(* CODESYS project IoDrvSoundDemo.project

Project tree, tasks and I/O mapping:
  Device : CODESYS Control Win V3, 3S - Smart Software Solutions GmbH, order no. 305021, version 3.5.9.0
    application Application
      libraries: Standard, * (System); Analyzation, * (System); IecSfc, * (System)
      task Task (cyclic, interval t#20ms, priority 1) calls Main_PRG
      program Main_PRG [ST]
      visualisation MainVisu
      Function Blocks/
        function block JukeBox [ST]
      Enums/
        data type STATE
      GlobalVariables/
        global variables HAENSCHEN_KLEIN
        global variables FUER_ELISE
        global variables X_MAX
        global variables MUSICAL_SYMBOLS
      Structs/
        data type NOTE
      VisElements/
        visualisation Piano
        visualisation JukeBox
        image pool ImagePool
    SoundCard : SoundCard, Sound Company, version 3.3.0.0
        output ding : BOOL  // SoundOutput.Byte0.Bit0
        output cord : BOOL  // SoundOutput.Byte0.Bit1
        output chimes : BOOL  // SoundOutput.Byte0.Bit2
        output notify : BOOL  // SoundOutput.Byte0.Bit3
        output ringout : BOOL  // SoundOutput.Byte0.Bit4
        output tada : BOOL  // SoundOutput.Byte0.Bit5
        output _type : BOOL  // SoundOutput.Byte0.Bit6
        output newmail : BOOL  // SoundOutput.Byte0.Bit7
        output C : BOOL  // SoundOutput.Byte1.Bit0
        output Cis : BOOL  // SoundOutput.Byte1.Bit1
        output D : BOOL  // SoundOutput.Byte1.Bit2
        output Dis : BOOL  // SoundOutput.Byte1.Bit3
        output E : BOOL  // SoundOutput.Byte1.Bit4
        output F : BOOL  // SoundOutput.Byte1.Bit5
        output Fis : BOOL  // SoundOutput.Byte1.Bit6
        output G : BOOL  // SoundOutput.Byte1.Bit7
        output Gis : BOOL  // SoundOutput.Byte2.Bit0
        output A : BOOL  // SoundOutput.Byte2.Bit1
        output Ais : BOOL  // SoundOutput.Byte2.Bit2
        output H : BOOL  // SoundOutput.Byte2.Bit3
        output C_ : BOOL  // SoundOutput.Byte2.Bit4
        output Cis_ : BOOL  // SoundOutput.Byte2.Bit5
        output D_ : BOOL  // SoundOutput.Byte2.Bit6
        output Dis_ : BOOL  // SoundOutput.Byte2.Bit7
        output E_ : BOOL  // SoundOutput.Byte3.Bit0
        output F_ : BOOL  // SoundOutput.Byte3.Bit1
        output Fis_ : BOOL  // SoundOutput.Byte3.Bit2
        output G_ : BOOL  // SoundOutput.Byte3.Bit3
        output Gis_ : BOOL  // SoundOutput.Byte3.Bit4
        output A_ : BOOL  // SoundOutput.Byte3.Bit5
        output Ais_ : BOOL  // SoundOutput.Byte3.Bit6
        output H_ : BOOL  // SoundOutput.Byte3.Bit7
        unmapped channels: SoundOutput
  text list GlobalTextList
  5ce3da45-db07-42e7-a21c-a00fff4ed8f6|files\Jukebox\Fifties_jukebox.png
  5ce3da45-db07-42e7-a21c-a00fff4ed8f6|files\Jukebox\Fifties_jukebox9.png
  5ce3da45-db07-42e7-a21c-a00fff4ed8f6|files\Jukebox\Fifties_jukebox10.png
  5ce3da45-db07-42e7-a21c-a00fff4ed8f6|files\Jukebox\Fifties_jukebox11.png
  5ce3da45-db07-42e7-a21c-a00fff4ed8f6|files\Jukebox\Fifties_jukebox12.png
  5ce3da45-db07-42e7-a21c-a00fff4ed8f6|files\Jukebox\Fifties_jukebox13.png
  5ce3da45-db07-42e7-a21c-a00fff4ed8f6|files\Jukebox\Fifties_jukebox_1.png
  5ce3da45-db07-42e7-a21c-a00fff4ed8f6|files\Jukebox\Fifties_jukebox_2.png
  5ce3da45-db07-42e7-a21c-a00fff4ed8f6|files\Jukebox\Fifties_jukebox3.png
  5ce3da45-db07-42e7-a21c-a00fff4ed8f6|files\Jukebox\Fifties_jukebox4.png
  5ce3da45-db07-42e7-a21c-a00fff4ed8f6|files\Jukebox\Fifties_jukebox5.png
  5ce3da45-db07-42e7-a21c-a00fff4ed8f6|files\Jukebox\Fifties_jukebox6.png
  5ce3da45-db07-42e7-a21c-a00fff4ed8f6|files\Jukebox\Fifties_jukebox7.png
  5ce3da45-db07-42e7-a21c-a00fff4ed8f6|files\Jukebox\Fifties_jukebox8.png
*)

// Device/Application/Enums/STATE
// Each value represents a state which the program can have
{attribute 'qualified_only'}
TYPE STATE :
(
	PIANO := 0,			// change to Piano mode
	MUTE,				// No sound will be played 
	FUER_ELISE,			// play 'Für Elise' from Ludwig van Beethoven
	HAENSCHEN_KLEIN,	// play 'Hänschen klein' a German folk song from Franz Wiedemann 
	MERRY_XMAS,			// play 'We Wish You a Merry Christmas' 
	JUKE,				// change to Jukebox mode
	WAITING				// waiting for another command
);
END_TYPE

// Device/Application/Structs/NOTE
// This structure represents a note that can be played by the program
TYPE NOTE :
STRUCT
	tLength	: TIME;				// reflects duration of a note
	pNote	: POINTER TO BYTE;	// byte address of the output channel
	iBit	: INT;				// Offset from the output byte that addresses the sound
END_STRUCT
END_TYPE

// Device/Application/GlobalVariables/HAENSCHEN_KLEIN
// Hänschen klein - Franz Wiedemann
VAR_GLOBAL
	HAENSCHEN : ARRAY[0..31] OF NOTE := [
		(************ Takt01 ***************************)
		(	tLength:= 	T#500MS ,
			pNote :=	ADR(IoConfig_Globals_Mapping.G),
			iBit	:= 7
		),
		(	tLength:= 	T#450MS ,
			pNote :=	ADR(IoConfig_Globals_Mapping.E),
			iBit	:= 4
		),
		(	tLength:= 	T#50MS ,
			pNote :=	ADR(MUSICAL_SYMBOLS.xPause),
			iBit	:= 0
		),
		(	tLength:= 	T#1000MS ,
			pNote :=	ADR(IoConfig_Globals_Mapping.E),
			iBit	:= 4
		),
		(************ Takt02 ***************************)
		(	tLength:= 	T#500MS ,
			pNote :=	ADR(IoConfig_Globals_Mapping.F),
			iBit	:= 5
		),
		(	tLength:= 	T#450MS ,
			pNote :=	ADR(IoConfig_Globals_Mapping.D),
			iBit	:= 2
		),
		(	tLength:= 	T#50MS ,
			pNote :=	ADR(MUSICAL_SYMBOLS.xPause),
			iBit	:= 0
		),
		(	tLength:= 	T#1000MS ,
			pNote :=	ADR(IoConfig_Globals_Mapping.D),
			iBit	:= 2
		),
		(************ Takt03 ***************************)
		(	tLength:= 	T#500MS ,
			pNote :=	ADR(IoConfig_Globals_Mapping.C),
			iBit	:= 0
		),
		(	tLength:= 	T#500MS ,
			pNote :=	ADR(IoConfig_Globals_Mapping.D),
			iBit	:= 2
		),
		(	tLength:= 	T#500MS ,
			pNote :=	ADR(IoConfig_Globals_Mapping.E),
			iBit	:= 4
		),
		(	tLength:= 	T#500MS ,
			pNote :=	ADR(IoConfig_Globals_Mapping.F),
			iBit	:= 5
		),
		(************ Takt04 ***************************)
		(	tLength:= 	T#450MS ,
			pNote :=	ADR(IoConfig_Globals_Mapping.G),
			iBit	:= 7
		),
		(	tLength:= 	T#50MS ,
			pNote :=	ADR(MUSICAL_SYMBOLS.xPause),
			iBit	:= 0
		),
		(	tLength:= 	T#450MS ,
			pNote :=	ADR(IoConfig_Globals_Mapping.G),
			iBit	:= 7
		),
		(	tLength:= 	T#50MS ,
			pNote :=	ADR(MUSICAL_SYMBOLS.xPause),
			iBit	:= 0
		),
		(	tLength:= 	T#1000MS ,
			pNote :=	ADR(IoConfig_Globals_Mapping.G),
			iBit	:= 7
		),
		(************ Takt05 ***************************)
		(	tLength:= 	T#50MS ,
			pNote :=	ADR(MUSICAL_SYMBOLS.xPause),
			iBit	:= 0
		),
		(	tLength:= 	T#450MS ,
			pNote :=	ADR(IoConfig_Globals_Mapping.G),
			iBit	:= 7
		),
		(	tLength:= 	T#450MS ,
			pNote :=	ADR(IoConfig_Globals_Mapping.E),
			iBit	:= 4
		),
		(	tLength:= 	T#50MS ,
			pNote :=	ADR(MUSICAL_SYMBOLS.xPause),
			iBit	:= 0
		),
		(	tLength:= 	T#1000MS ,
			pNote :=	ADR(IoConfig_Globals_Mapping.E),
			iBit	:= 4
		),
		(************ Takt06 ***************************)
		(	tLength:= 	T#500MS ,
			pNote :=	ADR(IoConfig_Globals_Mapping.F),
			iBit	:= 5
		),
		(	tLength:= 	T#450MS ,
			pNote :=	ADR(IoConfig_Globals_Mapping.D),
			iBit	:= 2
		),
		(	tLength:= 	T#50MS ,
			pNote :=	ADR(MUSICAL_SYMBOLS.xPause),
			iBit	:= 0
		),
		(	tLength:= 	T#1000MS ,
			pNote :=	ADR(IoConfig_Globals_Mapping.D),
			iBit	:= 2
		),
		(************ Takt07 ***************************)
		(	tLength:= 	T#500MS ,
			pNote :=	ADR(IoConfig_Globals_Mapping.C),
			iBit	:= 0
		),
		(	tLength:= 	T#500MS ,
			pNote :=	ADR(IoConfig_Globals_Mapping.E),
			iBit	:= 4
		),
		(	tLength:= 	T#450MS ,
			pNote :=	ADR(IoConfig_Globals_Mapping.G),
			iBit	:= 7
		),
		(	tLength:= 	T#50MS ,
			pNote :=	ADR(MUSICAL_SYMBOLS.xPause),
			iBit	:= 0
		),
		(	tLength:= 	T#500MS ,
			pNote :=	ADR(IoConfig_Globals_Mapping.G),
			iBit	:= 7
		),
		(************ Takt08 ***************************)
		(	tLength:= 	T#4000MS ,
			pNote :=	ADR(IoConfig_Globals_Mapping.C),
			iBit	:= 0
		)
	];
		
END_VAR

// Device/Application/GlobalVariables/FUER_ELISE
// Für Elise - Ludwig van Beethoven

VAR_GLOBAL
	ELISE : ARRAY[0..149] OF NOTE := [
		(************ Auftakt ***************************)
		(	tLength:= 	T#250MS ,
			pNote :=	ADR(IoConfig_Globals_Mapping.E_),
			iBit	:= 0
		),
		(	tLength:= 	T#250MS ,
			pNote :=	ADR(IoConfig_Globals_Mapping.Dis_),
			iBit	:= 7
		),
		(************ Takt01 ***************************)
		(	tLength:= 	T#250MS ,
			pNote :=	ADR(IoConfig_Globals_Mapping.E_),
			iBit	:= 0
		),
		(	tLength:= 	T#250MS ,
			pNote :=	ADR(IoConfig_Globals_Mapping.Dis_),
			iBit	:= 7
		),
		(	tLength:= 	T#250MS ,
			pNote :=	ADR(IoConfig_Globals_Mapping.E_),
			iBit	:= 0
		),
		(	tLength:= 	T#250MS ,
			pNote :=	ADR(IoConfig_Globals_Mapping.H),
			iBit	:= 3
		),
		(	tLength:= 	T#250MS ,
			pNote :=	ADR(IoConfig_Globals_Mapping.D_),
			iBit	:= 6
		),
		(	tLength:= 	T#250MS ,
			pNote :=	ADR(IoConfig_Globals_Mapping.C_),
			iBit	:= 4
		),
		(************ Takt02 ***************************)
		(	tLength:= 	T#500MS ,
			pNote :=	ADR(IoConfig_Globals_Mapping.A),
			iBit	:= 1
		),
		(	tLength:= 	T#250MS ,
			pNote :=	ADR(MUSICAL_SYMBOLS.xPause),
			iBit	:= 0
		),
		(	tLength:= 	T#250MS ,
			pNote :=	ADR(IoConfig_Globals_Mapping.C),
			iBit	:= 0
		),
		(	tLength:= 	T#250MS ,
			pNote :=	ADR(IoConfig_Globals_Mapping.E),
			iBit	:= 4
		),
		(	tLength:= 	T#250MS ,
			pNote :=	ADR(IoConfig_Globals_Mapping.A),
			iBit	:= 1
		),
		(************ Takt03 ***************************)
		(	tLength:= 	T#500MS ,
			pNote :=	ADR(IoConfig_Globals_Mapping.H),
			iBit	:= 3
		),
		(	tLength:= 	T#250MS ,
			pNote :=	ADR(MUSICAL_SYMBOLS.xPause),
			iBit	:= 0
		),
		(	tLength:= 	T#250MS ,
			pNote :=	ADR(IoConfig_Globals_Mapping.E),
			iBit	:= 4
		),
		(	tLength:= 	T#250MS ,
			pNote :=	ADR(IoConfig_Globals_Mapping.Gis),
			iBit	:= 0
		),
		(	tLength:= 	T#250MS ,
			pNote :=	ADR(IoConfig_Globals_Mapping.H),
			iBit	:= 3
		),
		(************ Takt04  ***************************)
		(	tLength:= 	T#500MS ,
			pNote :=	ADR(IoConfig_Globals_Mapping.C_),
			iBit	:= 4
		), 
		(	tLength:= 	T#250MS ,
			pNote :=	ADR(MUSICAL_SYMBOLS.xPause),
			iBit	:= 0
		),
		(	tLength:= 	T#250MS ,
			pNote :=	ADR(IoConfig_Globals_Mapping.E),
			iBit	:= 4
		),
		(	tLength:= 	T#250MS ,
			pNote :=	ADR(IoConfig_Globals_Mapping.E_),
			iBit	:= 0
		),
		(	tLength:= 	T#250MS ,
			pNote :=	ADR(IoConfig_Globals_Mapping.Dis_),
			iBit	:= 7
		),
		(************ Takt05 ***************************)
		(	tLength:= 	T#250MS ,
			pNote :=	ADR(IoConfig_Globals_Mapping.E_),
			iBit	:= 0
		),
		(	tLength:= 	T#250MS ,
			pNote :=	ADR(IoConfig_Globals_Mapping.Dis_),
			iBit	:= 7
		),
		(	tLength:= 	T#250MS ,
			pNote :=	ADR(IoConfig_Globals_Mapping.E_),
			iBit	:= 0
		),
		(	tLength:= 	T#250MS ,
			pNote :=	ADR(IoConfig_Globals_Mapping.H),
			iBit	:= 3
		),
		(	tLength:= 	T#250MS ,
			pNote :=	ADR(IoConfig_Globals_Mapping.D_),
			iBit	:= 6
		),
		(	tLength:= 	T#250MS ,
			pNote :=	ADR(IoConfig_Globals_Mapping.C_),
			iBit	:= 4
		),
		(************ Takt06 ***************************)
		(	tLength:= 	T#500MS ,
			pNote :=	ADR(IoConfig_Globals_Mapping.A),
			iBit	:= 1
		),
		(	tLength:= 	T#250MS ,
			pNote :=	ADR(MUSICAL_SYMBOLS.xPause),
			iBit	:= 0
		),
		(	tLength:= 	T#250MS ,
			pNote :=	ADR(IoConfig_Globals_Mapping.C),
			iBit	:= 0
		),
		(	tLength:= 	T#250MS ,
			pNote :=	ADR(IoConfig_Globals_Mapping.E),
			iBit	:= 4
		),
		(	tLength:= 	T#250MS ,
			pNote :=	ADR(IoConfig_Globals_Mapping.A),
			iBit	:= 1
		),
		(************ Takt07 ***************************)
		(	tLength:= 	T#500MS ,
			pNote :=	ADR(IoConfig_Globals_Mapping.H),
			iBit	:= 3
		),
		(	tLength:= 	T#50MS ,
			pNote :=	ADR(MUSICAL_SYMBOLS.xPause),
			iBit	:= 0
		),
		(	tLength:= 	T#200MS ,
			pNote :=	ADR(IoConfig_Globals_Mapping.E),
			iBit	:= 4
		),
		(	tLength:= 	T#250MS ,
			pNote :=	ADR(IoConfig_Globals_Mapping.C_),
			iBit	:= 4
		),
		(	tLength:= 	T#250MS ,
			pNote :=	ADR(IoConfig_Globals_Mapping.H),
			iBit	:= 3
		),
		(************ Takt08 ****************************)
		(	tLength:= 	T#1000MS ,
			pNote :=	ADR(IoConfig_Globals_Mapping.A),
			iBit	:= 1
		),
		(	tLength:= 	T#250MS ,
			pNote :=	ADR(IoConfig_Globals_Mapping.E_),
			iBit	:= 0
		),
		(	tLength:= 	T#250MS ,
			pNote :=	ADR(IoConfig_Globals_Mapping.Dis_),
			iBit	:= 7
		),
		(************ Takt09 ***************************)
		(	tLength:= 	T#250MS ,
			pNote :=	ADR(IoConfig_Globals_Mapping.E_),
			iBit	:= 0
		),
		(	tLength:= 	T#250MS ,
			pNote :=	ADR(IoConfig_Globals_Mapping.Dis_),
			iBit	:= 7
		),
		(	tLength:= 	T#250MS ,
			pNote :=	ADR(IoConfig_Globals_Mapping.E_),
			iBit	:= 0
		),
		(	tLength:= 	T#250MS ,
			pNote :=	ADR(IoConfig_Globals_Mapping.H),
			iBit	:= 3
		),
		(	tLength:= 	T#250MS ,
			pNote :=	ADR(IoConfig_Globals_Mapping.D_),
			iBit	:= 6
		),
		(	tLength:= 	T#250MS ,
			pNote :=	ADR(IoConfig_Globals_Mapping.C_),
			iBit	:= 4
		),
		(************ Takt10 ***************************)
		(	tLength:= 	T#500MS ,
			pNote :=	ADR(IoConfig_Globals_Mapping.A),
			iBit	:= 1
		),
		(	tLength:= 	T#250MS ,
			pNote :=	ADR(MUSICAL_SYMBOLS.xPause),
			iBit	:= 0
		),
		(	tLength:= 	T#250MS ,
			pNote :=	ADR(IoConfig_Globals_Mapping.C),
			iBit	:= 0
		),
		(	tLength:= 	T#250MS ,
			pNote :=	ADR(IoConfig_Globals_Mapping.E),
			iBit	:= 4
		),
		(	tLength:= 	T#250MS ,
			pNote :=	ADR(IoConfig_Globals_Mapping.A),
			iBit	:= 1
		),
		(************ Takt11 ***************************)
		(	tLength:= 	T#500MS ,
			pNote :=	ADR(IoConfig_Globals_Mapping.H),
			iBit	:= 3
		),
		(	tLength:= 	T#250MS ,
			pNote :=	ADR(MUSICAL_SYMBOLS.xPause),
			iBit	:= 0
		),
		(	tLength:= 	T#250MS ,
			pNote :=	ADR(IoConfig_Globals_Mapping.E),
			iBit	:= 4
		),
		(	tLength:= 	T#250MS ,
			pNote :=	ADR(IoConfig_Globals_Mapping.Gis),
			iBit	:= 0
		),
		(	tLength:= 	T#250MS ,
			pNote :=	ADR(IoConfig_Globals_Mapping.H),
			iBit	:= 3
		),
		(************ Takt12  ***************************)
		(	tLength:= 	T#500MS ,
			pNote :=	ADR(IoConfig_Globals_Mapping.C_),
			iBit	:= 4
		), 
		(	tLength:= 	T#250MS ,
			pNote :=	ADR(MUSICAL_SYMBOLS.xPause),
			iBit	:= 0
		),
		(	tLength:= 	T#250MS ,
			pNote :=	ADR(IoConfig_Globals_Mapping.E),
			iBit	:= 4
		),
		(	tLength:= 	T#250MS ,
			pNote :=	ADR(IoConfig_Globals_Mapping.E_),
			iBit	:= 0
		),
		(	tLength:= 	T#250MS ,
			pNote :=	ADR(IoConfig_Globals_Mapping.Dis_),
			iBit	:= 7
		),
		(************ Takt13 ***************************)
		(	tLength:= 	T#250MS ,
			pNote :=	ADR(IoConfig_Globals_Mapping.E_),
			iBit	:= 0
		),
		(	tLength:= 	T#250MS ,
			pNote :=	ADR(IoConfig_Globals_Mapping.Dis_),
			iBit	:= 7
		),
		(	tLength:= 	T#250MS ,
			pNote :=	ADR(IoConfig_Globals_Mapping.E_),
			iBit	:= 0
		),
		(	tLength:= 	T#250MS ,
			pNote :=	ADR(IoConfig_Globals_Mapping.H),
			iBit	:= 3
		),
		(	tLength:= 	T#250MS ,
			pNote :=	ADR(IoConfig_Globals_Mapping.D_),
			iBit	:= 6
		),
		(	tLength:= 	T#250MS ,
			pNote :=	ADR(IoConfig_Globals_Mapping.C_),
			iBit	:= 4
		),
		(************ Takt14 ***************************)
		(	tLength:= 	T#500MS ,
			pNote :=	ADR(IoConfig_Globals_Mapping.A),
			iBit	:= 1
		),
		(	tLength:= 	T#250MS ,
			pNote :=	ADR(MUSICAL_SYMBOLS.xPause),
			iBit	:= 0
		),
		(	tLength:= 	T#250MS ,
			pNote :=	ADR(IoConfig_Globals_Mapping.C),
			iBit	:= 0
		),
		(	tLength:= 	T#250MS ,
			pNote :=	ADR(IoConfig_Globals_Mapping.E),
			iBit	:= 4
		),
		(	tLength:= 	T#250MS ,
			pNote :=	ADR(IoConfig_Globals_Mapping.A),
			iBit	:= 1
		),
		(************ Takt15 ***************************)
		(	tLength:= 	T#500MS ,
			pNote :=	ADR(IoConfig_Globals_Mapping.H),
			iBit	:= 3
		),
		(	tLength:= 	T#50MS ,
			pNote :=	ADR(MUSICAL_SYMBOLS.xPause),
			iBit	:= 0
		),
		(	tLength:= 	T#200MS ,
			pNote :=	ADR(IoConfig_Globals_Mapping.E),
			iBit	:= 4
		),
		(	tLength:= 	T#250MS ,
			pNote :=	ADR(IoConfig_Globals_Mapping.C_),
			iBit	:= 4
		),
		(	tLength:= 	T#250MS ,
			pNote :=	ADR(IoConfig_Globals_Mapping.H),
			iBit	:= 3
		),
		(************ Takt16 ***************************)
		(	tLength:= 	T#500MS ,
			pNote :=	ADR(IoConfig_Globals_Mapping.A),
			iBit	:= 1
		),
		(	tLength:= 	T#250MS ,
			pNote :=	ADR(MUSICAL_SYMBOLS.xPause),
			iBit	:= 0
		),
		(	tLength:= 	T#200MS ,
			pNote :=	ADR(IoConfig_Globals_Mapping.H),
			iBit	:= 3
		),
		(	tLength:= 	T#250MS ,
			pNote :=	ADR(IoConfig_Globals_Mapping.C_),
			iBit	:= 4
		),
		(	tLength:= 	T#250MS ,
			pNote :=	ADR(IoConfig_Globals_Mapping.D_),
			iBit	:= 6
		),
		(************ Takt17  ***************************)
		(	tLength:= 	T#750MS ,
			pNote :=	ADR(IoConfig_Globals_Mapping.E_),
			iBit	:= 0
		),
		(	tLength:= 	T#250MS ,
			pNote :=	ADR(IoConfig_Globals_Mapping.G),
			iBit	:= 7
		),
		(	tLength:= 	T#250MS ,
			pNote :=	ADR(IoConfig_Globals_Mapping.F_),
			iBit	:= 1
		),
		(	tLength:= 	T#250MS ,
			pNote :=	ADR(IoConfig_Globals_Mapping.E_),
			iBit	:= 0
		),
		(************ Takt18 ***************************)
		(	tLength:= 	T#750MS ,
			pNote :=	ADR(IoConfig_Globals_Mapping.D_),
			iBit	:= 6
		),
		(	tLength:= 	T#250MS ,
			pNote :=	ADR(IoConfig_Globals_Mapping.F),
			iBit	:= 5
		),
		(	tLength:= 	T#250MS ,
			pNote :=	ADR(IoConfig_Globals_Mapping.E_),
			iBit	:= 0
		),
		(	tLength:= 	T#250MS ,
			pNote :=	ADR(IoConfig_Globals_Mapping.D_),
			iBit	:= 6
		),
		(************ Takt19 ***************************)
		(	tLength:= 	T#750MS ,
			pNote :=	ADR(IoConfig_Globals_Mapping.C_),
			iBit	:= 4
		),
		(	tLength:= 	T#250MS ,
			pNote :=	ADR(IoConfig_Globals_Mapping.E),
			iBit	:= 0
		),
		(	tLength:= 	T#250MS ,
			pNote :=	ADR(IoConfig_Globals_Mapping.D_),
			iBit	:= 6
		),
		(	tLength:= 	T#250MS ,
			pNote :=	ADR(IoConfig_Globals_Mapping.C_),
			iBit	:= 4
		),
		(************ Takt20 ***************************)
		(	tLength:= 	T#500MS ,
			pNote :=	ADR(IoConfig_Globals_Mapping.H),
			iBit	:= 3
		),
		(	tLength:= 	T#250MS ,
			pNote :=	ADR(MUSICAL_SYMBOLS.xPause),
			iBit	:= 0
		),
		(	tLength:= 	T#250MS ,
			pNote :=	ADR(IoConfig_Globals_Mapping.E),
			iBit	:= 4
		),
		(	tLength:= 	T#250MS ,
			pNote :=	ADR(IoConfig_Globals_Mapping.E_),
			iBit	:= 0
		),
		(	tLength:= 	T#250MS ,
			pNote :=	ADR(MUSICAL_SYMBOLS.xPause),
			iBit	:= 0
		),
		(************ Takt21 ***************************)
		(	tLength:= 	T#250MS ,
			pNote :=	ADR(MUSICAL_SYMBOLS.xPause),
			iBit	:= 0
		),
		(	tLength:= 	T#250MS ,
			pNote :=	ADR(IoConfig_Globals_Mapping.E_),
			iBit	:= 0
		),
		(	tLength:= 	T#250MS ,
			pNote :=	ADR(IoConfig_Globals_Mapping.E),
			iBit	:= 4
		),
		(	tLength:= 	T#500MS ,
			pNote :=	ADR(MUSICAL_SYMBOLS.xPause),
			iBit	:= 0
		),
		(	tLength:= 	T#250MS ,
			pNote :=	ADR(IoConfig_Globals_Mapping.Dis_),
			iBit	:= 7
		),
		(************ Takt22 ***************************)
		(	tLength:= 	T#250MS ,
			pNote :=	ADR(IoConfig_Globals_Mapping.E_),
			iBit	:= 0
		),
		(	tLength:= 	T#500MS ,
			pNote :=	ADR(MUSICAL_SYMBOLS.xPause),
			iBit	:= 0
		),
		(	tLength:= 	T#250MS ,
			pNote :=	ADR(IoConfig_Globals_Mapping.Dis_),
			iBit	:= 7
		),
		(	tLength:= 	T#250MS ,
			pNote :=	ADR(IoConfig_Globals_Mapping.E_),
			iBit	:= 0
		),
		(	tLength:= 	T#250MS ,
			pNote :=	ADR(IoConfig_Globals_Mapping.D_),
			iBit	:= 6
		),
		(************ Takt23 ***************************)
		(	tLength:= 	T#250MS ,
			pNote :=	ADR(IoConfig_Globals_Mapping.E_),
			iBit	:= 0
		),
		(	tLength:= 	T#250MS ,
			pNote :=	ADR(IoConfig_Globals_Mapping.Dis_),
			iBit	:= 7
		),
		(	tLength:= 	T#250MS ,
			pNote :=	ADR(IoConfig_Globals_Mapping.E_),
			iBit	:= 0
		),
		(	tLength:= 	T#250MS ,
			pNote :=	ADR(IoConfig_Globals_Mapping.H),
			iBit	:= 3
		),
		(	tLength:= 	T#250MS ,
			pNote :=	ADR(IoConfig_Globals_Mapping.D_),
			iBit	:= 6
		),
		(	tLength:= 	T#250MS ,
			pNote :=	ADR(IoConfig_Globals_Mapping.C_),
			iBit	:= 4
		),
		(************ Takt24 ***************************)
		(	tLength:= 	T#500MS ,
			pNote :=	ADR(IoConfig_Globals_Mapping.A),
			iBit	:= 1
		),
		(	tLength:= 	T#250MS ,
			pNote :=	ADR(MUSICAL_SYMBOLS.xPause),
			iBit	:= 0
		),
		(	tLength:= 	T#250MS ,
			pNote :=	ADR(IoConfig_Globals_Mapping.C),
			iBit	:= 0
		),
		(	tLength:= 	T#250MS ,
			pNote :=	ADR(IoConfig_Globals_Mapping.E),
			iBit	:= 4
		),
		(	tLength:= 	T#250MS ,
			pNote :=	ADR(IoConfig_Globals_Mapping.A),
			iBit	:= 1
		),
		(************ Takt25 ***************************)
		(	tLength:= 	T#500MS ,
			pNote :=	ADR(IoConfig_Globals_Mapping.H),
			iBit	:= 3
		),
		(	tLength:= 	T#250MS ,
			pNote :=	ADR(MUSICAL_SYMBOLS.xPause),
			iBit	:= 0
		),
		(	tLength:= 	T#250MS ,
			pNote :=	ADR(IoConfig_Globals_Mapping.E),
			iBit	:= 4
		),
		(	tLength:= 	T#250MS ,
			pNote :=	ADR(IoConfig_Globals_Mapping.Gis),
			iBit	:= 0
		),
		(	tLength:= 	T#250MS ,
			pNote :=	ADR(IoConfig_Globals_Mapping.H),
			iBit	:= 3
		),
		(************ Takt26  ***************************)
		(	tLength:= 	T#500MS ,
			pNote :=	ADR(IoConfig_Globals_Mapping.C_),
			iBit	:= 4
		), 
		(	tLength:= 	T#250MS ,
			pNote :=	ADR(MUSICAL_SYMBOLS.xPause),
			iBit	:= 0
		),
		(	tLength:= 	T#250MS ,
			pNote :=	ADR(IoConfig_Globals_Mapping.E),
			iBit	:= 4
		),
		(	tLength:= 	T#250MS ,
			pNote :=	ADR(IoConfig_Globals_Mapping.E_),
			iBit	:= 0
		),
		(	tLength:= 	T#250MS ,
			pNote :=	ADR(IoConfig_Globals_Mapping.Dis_),
			iBit	:= 7
		),
		(************ Takt27 ***************************)
		(	tLength:= 	T#250MS ,
			pNote :=	ADR(IoConfig_Globals_Mapping.E_),
			iBit	:= 0
		),
		(	tLength:= 	T#250MS ,
			pNote :=	ADR(IoConfig_Globals_Mapping.Dis_),
			iBit	:= 7
		),
		(	tLength:= 	T#250MS ,
			pNote :=	ADR(IoConfig_Globals_Mapping.E_),
			iBit	:= 0
		),
		(	tLength:= 	T#250MS ,
			pNote :=	ADR(IoConfig_Globals_Mapping.H),
			iBit	:= 3
		),
		(	tLength:= 	T#250MS ,
			pNote :=	ADR(IoConfig_Globals_Mapping.D_),
			iBit	:= 6
		),
		(	tLength:= 	T#250MS ,
			pNote :=	ADR(IoConfig_Globals_Mapping.C_),
			iBit	:= 4
		),
		(************ Takt28 ***************************)
		(	tLength:= 	T#500MS ,
			pNote :=	ADR(IoConfig_Globals_Mapping.A),
			iBit	:= 1
		),
		(	tLength:= 	T#250MS ,
			pNote :=	ADR(MUSICAL_SYMBOLS.xPause),
			iBit	:= 0
		),
		(	tLength:= 	T#250MS ,
			pNote :=	ADR(IoConfig_Globals_Mapping.C),
			iBit	:= 0
		),
		(	tLength:= 	T#250MS ,
			pNote :=	ADR(IoConfig_Globals_Mapping.E),
			iBit	:= 4
		),
		(	tLength:= 	T#250MS ,
			pNote :=	ADR(IoConfig_Globals_Mapping.A),
			iBit	:= 1
		),
		(************ Takt29 ***************************)
		(	tLength:= 	T#500MS ,
			pNote :=	ADR(IoConfig_Globals_Mapping.H),
			iBit	:= 3
		),
		(	tLength:= 	T#50MS ,
			pNote :=	ADR(MUSICAL_SYMBOLS.xPause),
			iBit	:= 0
		),
		(	tLength:= 	T#200MS ,
			pNote :=	ADR(IoConfig_Globals_Mapping.E),
			iBit	:= 4
		),
		(	tLength:= 	T#250MS ,
			pNote :=	ADR(IoConfig_Globals_Mapping.C_),
			iBit	:= 4
		),
		(	tLength:= 	T#250MS ,
			pNote :=	ADR(IoConfig_Globals_Mapping.H),
			iBit	:= 3
		),
		(************ Takt30 ****************************)
		(	tLength:= 	T#500MS ,
			pNote :=	ADR(IoConfig_Globals_Mapping.A),
			iBit	:= 1
		),
		(	tLength:= 	T#1000MS ,
			pNote :=	ADR(MUSICAL_SYMBOLS.xPause),
			iBit	:= 1
		)
	
		];
		
END_VAR

// Device/Application/GlobalVariables/X_MAX
// We Wish You a Merry Christmas
VAR_GLOBAL
	XMAS : ARRAY[0..36] OF NOTE := [
		(************ Auftakt ***************************)
		(	tLength:= 	T#500MS ,
			pNote :=	ADR(IoConfig_Globals_Mapping.G),
			iBit	:= 7
		),
		(************ Takt01 ***************************)
		(	tLength:= 	T#450MS ,
			pNote :=	ADR(IoConfig_Globals_Mapping.C_),
			iBit	:= 4
		),
		(	tLength:= 	T#50MS ,
			pNote :=	ADR(MUSICAL_SYMBOLS.xPause),
			iBit	:= 0
		),
		(	tLength:= 	T#250MS ,
			pNote :=	ADR(IoConfig_Globals_Mapping.C_),
			iBit	:= 4
		),
		(	tLength:= 	T#250MS ,
			pNote :=	ADR(IoConfig_Globals_Mapping.D_),
			iBit	:= 6
		),
		(	tLength:= 	T#250MS ,
			pNote :=	ADR(IoConfig_Globals_Mapping.C_),
			iBit	:= 4
		),
		(	tLength:= 	T#250MS ,
			pNote :=	ADR(IoConfig_Globals_Mapping.H),
			iBit	:= 3
		),
		(************ Takt02 ***************************)
		(	tLength:= 	T#450MS ,
			pNote :=	ADR(IoConfig_Globals_Mapping.A),
			iBit	:= 1
		),
		(	tLength:= 	T#50MS ,
			pNote :=	ADR(MUSICAL_SYMBOLS.xPause),
			iBit	:= 0
		),
		(	tLength:= 	T#450MS ,
			pNote :=	ADR(IoConfig_Globals_Mapping.A),
			iBit	:= 1
		),
		(	tLength:= 	T#50MS ,
			pNote :=	ADR(MUSICAL_SYMBOLS.xPause),
			iBit	:= 0
		),
		(	tLength:= 	T#500MS ,
			pNote :=	ADR(IoConfig_Globals_Mapping.A),
			iBit	:= 1
		),
		(************ Takt03 ***************************)
		(	tLength:= 	T#450MS ,
			pNote :=	ADR(IoConfig_Globals_Mapping.D_),
			iBit	:= 6
		),
		(	tLength:= 	T#50MS ,
			pNote :=	ADR(MUSICAL_SYMBOLS.xPause),
			iBit	:= 0
		),
		(	tLength:= 	T#250MS ,
			pNote :=	ADR(IoConfig_Globals_Mapping.D_),
			iBit	:= 6
		),
		(	tLength:= 	T#250MS ,
			pNote :=	ADR(IoConfig_Globals_Mapping.E_),
			iBit	:= 0
		),
		(	tLength:= 	T#250MS ,
			pNote :=	ADR(IoConfig_Globals_Mapping.D_),
			iBit	:= 6
		),
		(	tLength:= 	T#250MS ,
			pNote :=	ADR(IoConfig_Globals_Mapping.C_),
			iBit	:= 4
		),
		(************ Takt04 ***************************)
		(	tLength:= 	T#500MS ,
			pNote :=	ADR(IoConfig_Globals_Mapping.H),
			iBit	:= 3
		),
		(	tLength:= 	T#450MS ,
			pNote :=	ADR(IoConfig_Globals_Mapping.G),
			iBit	:= 7
		),
		(	tLength:= 	T#50MS ,
			pNote :=	ADR(MUSICAL_SYMBOLS.xPause),
			iBit	:= 0
		),
		(	tLength:= 	T#500MS ,
			pNote :=	ADR(IoConfig_Globals_Mapping.G),
			iBit	:= 7
		),
		(************ Takt05 ***************************)
		(	tLength:= 	T#450MS ,
			pNote :=	ADR(IoConfig_Globals_Mapping.E_),
			iBit	:= 0
		),
		(	tLength:= 	T#50MS ,
			pNote :=	ADR(MUSICAL_SYMBOLS.xPause),
			iBit	:= 0
		),
		(	tLength:= 	T#250MS ,
			pNote :=	ADR(IoConfig_Globals_Mapping.E_),
			iBit	:= 0
		),
		(	tLength:= 	T#250MS ,
			pNote :=	ADR(IoConfig_Globals_Mapping.F_),
			iBit	:= 1
		),
		(	tLength:= 	T#250MS ,
			pNote :=	ADR(IoConfig_Globals_Mapping.E_),
			iBit	:= 0
		),
		(	tLength:= 	T#250MS ,
			pNote :=	ADR(IoConfig_Globals_Mapping.D_),
			iBit	:= 6
		),
		(************ Takt06 ***************************)
		(	tLength:= 	T#500MS ,
			pNote :=	ADR(IoConfig_Globals_Mapping.C_),
			iBit	:= 4
		),
		(	tLength:= 	T#500MS ,
			pNote :=	ADR(IoConfig_Globals_Mapping.A),
			iBit	:= 1
		),
		(	tLength:= 	T#250MS ,
			pNote :=	ADR(IoConfig_Globals_Mapping.G),
			iBit	:= 7
		),
		(	tLength:= 	T#50MS ,
			pNote :=	ADR(MUSICAL_SYMBOLS.xPause),
			iBit	:= 0
		),
		(	tLength:= 	T#200MS ,
			pNote :=	ADR(IoConfig_Globals_Mapping.G),
			iBit	:= 7
		),
		(************ Takt07 ***************************)
		(	tLength:= 	T#500MS ,
			pNote :=	ADR(IoConfig_Globals_Mapping.A),
			iBit	:= 1
		),
		(	tLength:= 	T#500MS ,
			pNote :=	ADR(IoConfig_Globals_Mapping.D_),
			iBit	:= 6
		),
		(	tLength:= 	T#500MS ,
			pNote :=	ADR(IoConfig_Globals_Mapping.H),
			iBit	:= 3
		),
		(************ Takt07 ***************************)
		(	tLength:= 	T#1000MS ,
			pNote :=	ADR(IoConfig_Globals_Mapping.C_),
			iBit	:= 4
		)
		];
END_VAR

// Device/Application/GlobalVariables/MUSICAL_SYMBOLS
{attribute 'qualified_only'}
VAR_GLOBAL
	xPause	: BOOL;
END_VAR

// Device/Application/Main_PRG
/// This example demos the mapping of outputs. For illustration it uses a sound card and a program that
/// allows the user to play some music.
/// The Sound Demo Main_PRG contains the main logic behind this example
/// it constantly changes between seven different states (see STATE enumeration for more information).
/// This Program offers a Piano with the great and small octave.
/// There is also a Jukebox Mode where the user can play three different songs. 
	 
PROGRAM Main_PRG
VAR
	eState		: STATE := STATE.PIANO;	(* holds the current state of the program *)
	xPlayPiano	: BOOL;					(* if true the Piano will be visible in MainVisu *)
	xPlayJuke	: BOOL;					(* if true the Jukebox will be visible in MainVisu *)

	iCnt		: INT;					(* contains the length of a song *)
	iBit		: INT;					(* offset from the output byte *)
	Timer		: TON;					(* manages the sound length *)
	
	pbyNote		: POINTER TO BYTE;		(* output byte *)
	Jukebox		: Jukebox;				(* Function Block for jukebox animation *)
	xPlay		: BOOL := TRUE;			(* TRUE starts the music program *)
END_VAR

VAR_INPUT
END_VAR
VAR_OUTPUT
END_VAR

IF xPlay THEN
	
	CASE eState OF
		STATE.MUTE: (* set all output bits to false and stop playing a sound *)
				Jukebox(xStart:=FALSE);
				
				C := FALSE;
				Cis := FALSE;
				D := FALSE;
				Dis := FALSE;
				E := FALSE;
				F := FALSE;
				Fis := FALSE;
				G := FALSE;
				Gis := FALSE;
				A := FALSE;
				Ais := FALSE;
				H := FALSE;
				C_ := FALSE;
				Cis_ := FALSE;
				D_ := FALSE;
				Dis_ := FALSE;
				E_ := FALSE;
				F_ := FALSE;
				Fis_ := FALSE;
				G_ := FALSE;
				Gis_ := FALSE;
				A_ := FALSE;
				Ais_ := FALSE;
				H_ := FALSE;
				
				eState:= STATE.WAITING;
				
		STATE.FUER_ELISE: (* start playing 'Für Elise' *)
				Jukebox(xStart:=TRUE);
				IF iCnt <= 149 THEN
					Timer(in:=TRUE, pt:=ELISE[iCnt].tLength, Q=>);
					iBit:= ELISE[iCnt].iBit;
					pbyNote:=ELISE[iCnt].pNote;
					pbyNote^:=SHL(1,ELISE[iCnt].iBit);
					IF Timer.Q THEN
						Timer(in:=FALSE);
						pbyNote^:=SHL(0,ELISE[iCnt].iBit);
						iCnt:=iCnt+1;
					END_IF
				ELSE
					iCnt:=0;
				END_IF
				
		STATE.HAENSCHEN_KLEIN: (* start playing 'Hänschen klein' *)
				Jukebox(xStart:=TRUE);
				IF iCnt <= 31 THEN
					Timer(in:=TRUE, pt:=HAENSCHEN[iCnt].tLength, Q=>);
					iBit:= HAENSCHEN[iCnt].iBit;
					pbyNote:=HAENSCHEN[iCnt].pNote;
					pbyNote^:=SHL(1,HAENSCHEN[iCnt].iBit);
					IF Timer.Q THEN
						Timer(in:=FALSE);
						pbyNote^:=SHL(0,HAENSCHEN[iCnt].iBit);
						iCnt:=iCnt+1;
					END_IF
				ELSE
					iCnt:=0;
				END_IF
				
				
		STATE.MERRY_XMAS: (* start playing 'We Wish You a Merry Christmas' *)
				Jukebox(xStart:=TRUE);
				IF iCnt <= 36 THEN
					Timer(in:=TRUE, pt:=XMAS[iCnt].tLength, Q=>);
					iBit:= XMAS[iCnt].iBit;
					pbyNote:=XMAS[iCnt].pNote;
					pbyNote^:=SHL(1,XMAS[iCnt].iBit);
					IF Timer.Q THEN
						Timer(in:=FALSE);
						pbyNote^:=SHL(0,XMAS[iCnt].iBit);
						iCnt:=iCnt+1;
					END_IF
				ELSE
					iCnt:=0;
				END_IF
	
				
		STATE.PIANO: (* change to Piano mode *)
				xPlayPiano := TRUE;
				xPlayJuke := FALSE;
				eState:=STATE.MUTE;
				
		STATE.JUKE: (* change to Jukebox mode *)
				xPlayPiano := FALSE;
				xPlayJuke := TRUE;
				eState:=STATE.MUTE;
				
		STATE.WAITING: (* wait for input from user *)
							
	END_CASE
END_IF

END_PROGRAM

// Device/Application/Function Blocks/JukeBox
/// The JukeBox FB controls the 'blinking' of the JukeBox in
/// the MainVisu. The Jukebox will change its appearance every 600ms. 
/// The cycle contains 13 different picture changes. 

{attribute 'hide_all_locals'}
FUNCTION_BLOCK JukeBox
VAR_INPUT
	xStart	: BOOL; (* If TRUE, the Jukebox starts to blink *)
END_VAR
VAR_OUTPUT
END_VAR
VAR
	iCnt	: INT; (* Counter *)
	xBling	: ARRAY[0..13] OF BOOL := [FALSE, 13(TRUE)]; (* This array holds the information whether a Jukebox picture is visible or not *)
	Timer	: ton; (* Timer for the image change *)
END_VAR

IF xStart THEN
	Timer(in:=xStart, pt:= T#600MS);
	xBling[iCnt] := FALSE;
	IF iCnt > 0 THEN
		xBling[iCnt-1] := TRUE;
	ELSIF iCnt = 0 THEN
		xBling[13] := TRUE;
	END_IF
	
	IF Timer.Q THEN
		iCnt:=iCnt+1;
		IF iCnt >13 THEN
			iCnt:=0;
		END_IF
		Timer(in:=FALSE);
	END_IF
END_IF

END_FUNCTION_BLOCK

// Device/Application/MainVisu
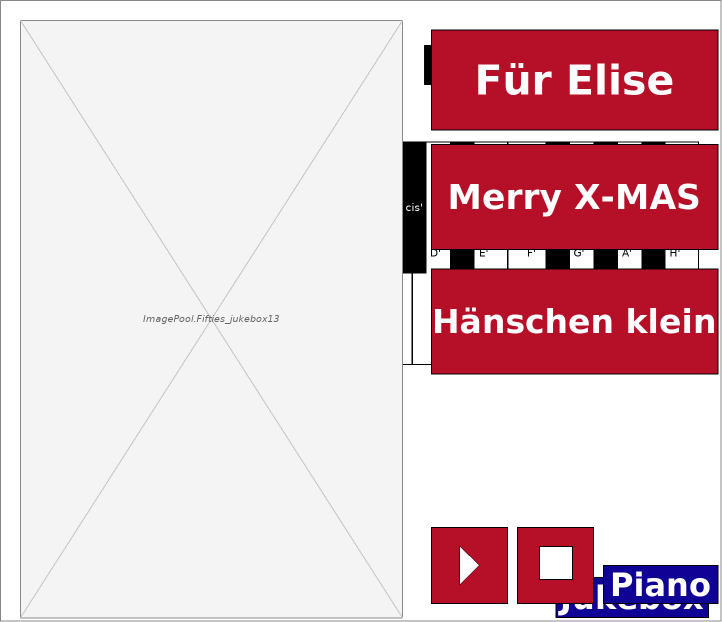
VISUALIZATION MainVisu  // 722x622
    Frame (20,20 700x600), invisible if: Main_PRG.xPlayJuke, input disabled if: Main_PRG.xPlayJuke
        shows Piano()
    Frame (20,20 700x600), invisible if: Main_PRG.xPlayPiano, input disabled if: Main_PRG.xPlayPiano
        shows JukeBox()
END_VISUALIZATION

// Device/Application/VisElements/Piano
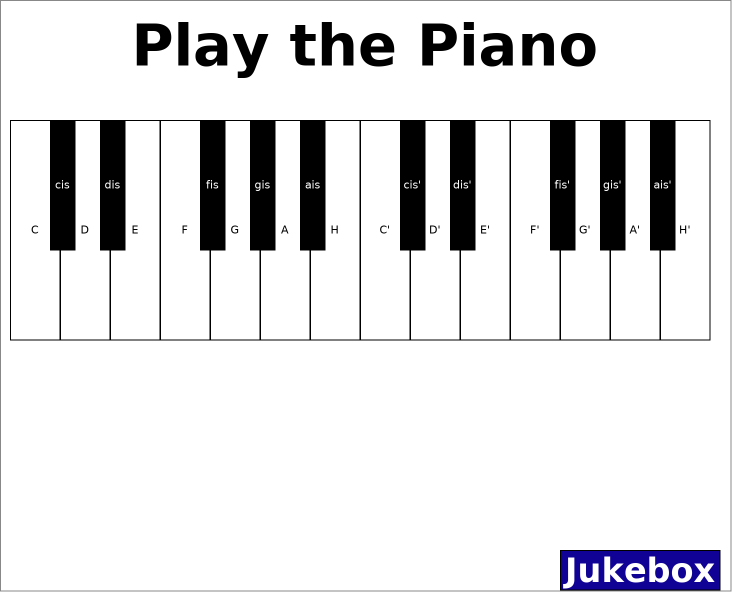
VISUALIZATION Piano  // 732x592
    Rectangle (10,130 350x140)
    RoundedRectangle (310,120 50x220), "H", colour toggle: H
        tap H
    RoundedRectangle (260,120 50x220), "A", colour toggle: A
        tap A
    RoundedRectangle (210,120 50x220), "G", colour toggle: G
        tap G
    RoundedRectangle (10,120 50x220), "C", colour toggle: C
        tap C
    RoundedRectangle (60,120 50x220), "D", colour toggle: D
        tap D
    RoundedRectangle (110,120 50x220), "E", colour toggle: E
        tap E
    RoundedRectangle (160,120 50x220), "F", colour toggle: F
        tap F
    Rectangle (300,120 25x130), "ais", colour toggle: Ais
        tap Ais
    Rectangle (250,120 25x130), "gis", colour toggle: Gis
        tap Gis
    Rectangle (200,120 25x130), "fis", colour toggle: Fis
        tap Fis
    Rectangle (100,120 25x130), "dis", colour toggle: Dis
        tap Dis
    Rectangle (50,120 25x130), "cis", colour toggle: Cis
        tap Cis
    RoundedRectangle (660,120 50x220), "H'", colour toggle: H_
        tap H_
    RoundedRectangle (610,120 50x220), "A'", colour toggle: A_
        tap A_
    RoundedRectangle (560,120 50x220), "G'", colour toggle: G_
        tap G_
    RoundedRectangle (360,120 50x220), "C'", colour toggle: C_
        tap C_
    RoundedRectangle (410,120 50x220), "D'", colour toggle: D_
        tap D_
    RoundedRectangle (460,120 50x220), "E'", colour toggle: E_
        tap E_
    RoundedRectangle (510,120 50x220), "F'", colour toggle: F_
        tap F_
    Rectangle (650,120 25x130), "ais'", colour toggle: Ais_
        tap Ais_
    Rectangle (600,120 25x130), "gis'", colour toggle: Gis_
        tap Gis_
    Rectangle (550,120 25x130), "fis'", colour toggle: Fis_
        tap Fis_
    Rectangle (450,120 25x130), "dis'", colour toggle: Dis_
        tap Dis_
    Rectangle (400,120 25x130), "cis'", colour toggle: Cis_
        tap Cis_
    Rectangle (560,550 160x40), "Jukebox"
        OnMouseClick: execute { Main_PRG.eState:=STATE.JUKE; }
    Label (0,10 730x70), "Play the Piano"
END_VISUALIZATION

// Device/Application/VisElements/JukeBox
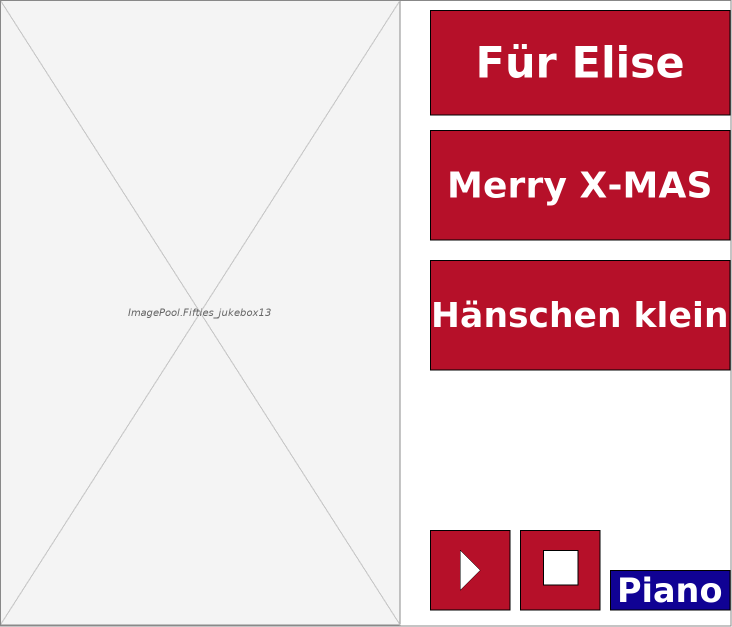
VISUALIZATION JukeBox  // 732x627
    Rectangle (430,530 80x80)
        OnMouseClick: execute { Main_PRG.xPlay:=false; }
    Rectangle (460,550 5x40)
        OnMouseClick: execute { Main_PRG.xPlay:=false; }
    Rectangle (480,550 5x40)
        OnMouseClick: execute { Main_PRG.xPlay:=false; }
    Image (0,0 400x625), invisible if: Main_PRG.Jukebox.xBling[0], image: ImagePool.JukeBoxOrg
    Image (0,0 400x625), invisible if: Main_PRG.Jukebox.xBling[1], image: ImagePool.Fifties_jukebox_1
    Image (0,0 400x625), invisible if: Main_PRG.Jukebox.xBling[2], image: ImagePool.Fifties_jukebox_2
    Image (0,0 400x625), invisible if: Main_PRG.Jukebox.xBling[3], image: ImagePool.Fifties_jukebox3
    Image (0,0 400x625), invisible if: Main_PRG.Jukebox.xBling[4], image: ImagePool.Fifties_jukebox4
    Image (0,0 400x625), invisible if: Main_PRG.Jukebox.xBling[5], image: ImagePool.Fifties_jukebox5
    Image (0,0 400x625), invisible if: Main_PRG.Jukebox.xBling[6], image: ImagePool.Fifties_jukebox6
    Image (0,0 400x625), invisible if: Main_PRG.Jukebox.xBling[7], image: ImagePool.Fifties_jukebox7
    Image (0,0 400x625), invisible if: Main_PRG.Jukebox.xBling[8], image: ImagePool.Fifties_jukebox8
    Image (0,0 400x625), invisible if: Main_PRG.Jukebox.xBling[9], image: ImagePool.Fifties_jukebox9
    Image (0,0 400x625), invisible if: Main_PRG.Jukebox.xBling[10], image: ImagePool.Fifties_jukebox10
    Image (0,0 400x625), invisible if: Main_PRG.Jukebox.xBling[11], image: ImagePool.Fifties_jukebox11
    Image (0,0 400x625), invisible if: Main_PRG.Jukebox.xBling[12], image: ImagePool.Fifties_jukebox12
    Image (0,0 400x625), invisible if: Main_PRG.Jukebox.xBling[13], image: ImagePool.Fifties_jukebox13
    Rectangle (430,10 300x105), "Für Elise"
        OnMouseClick: execute { Main_PRG.iCnt:=0; Main_PRG.eState:= STATE.FUER_ELISE; }
    Rectangle (430,130 300x110), "Merry X-MAS"
        OnMouseClick: execute { Main_PRG.iCnt:=0; Main_PRG.eState:= STATE.MERRY_XMAS; }
    Rectangle (430,260 300x110), "Hänschen klein"
        OnMouseClick: execute { Main_PRG.iCnt:=0; Main_PRG.eState:=STATE.HAENSCHEN_KLEIN; }
    Rectangle (520,530 80x80)
        OnMouseClick: execute { Main_PRG.eState:=STATE.JUKE; }
    Rectangle (610,570 120x40), "Piano"
        OnMouseClick: execute { Main_PRG.eState:=STATE.PIANO; }
    Rectangle (543,550 35x35)
        OnMouseClick: execute { Main_PRG.eState:=STATE.JUKE; }
    Rectangle (430,530 80x80), invisible if: Main_PRG.xPlay
        OnMouseClick: execute { Main_PRG.xPlay:=true; }
    Polygon (460,590) (460,550) (480,570), invisible if: Main_PRG.xPlay
        OnMouseClick: execute { Main_PRG.xPlay:=true; }
END_VISUALIZATION
